PROGRAM POU_SetStatus
VAR
END_VAR

END_PROGRAM

(* stored: Version 1.1.0.1, ProductVersion 3.1.4022.18
   POU POU_SetStatus: Id {04dac471-e342-4348-a3f6-e1eada599089}, SpecialFunc None *)
